// TIA Portal V20 export
// export: Created 2025-12-01T14:57:04.1801428Z, ExportSetting None, DisplayName Totally Integrated Automation Portal, DisplayVersion V20 Update 3, DisplayName TIA Portal Openness, DisplayVersion V20 Update 3, DisplayName TIA Portal Version Control Interface, DisplayVersion V20 Update 3, DisplayName STEP 7 Professional, DisplayVersion V20 Update 3, DisplayName STEP 7 Safety, DisplayVersion V20 Update 2, DisplayName WinCC Basic/Comfort/Advanced, DisplayVersion V20 Update 3, DisplayName WinCC Professional, DisplayVersion V20 Update 3, DisplayName WinCC Unified, DisplayVersion V20 Update 3
FUNCTION "FC762_EventosAlturaPedido" : Void   // FC762, STL
TITLE = Emision de los Eventos del la Etiquetadora
{ S7_Optimized_Access := 'FALSE' }
AUTHOR : TRACKING
NAME : 20141014
VERSION : 4.0
// stored: AutoNumber false
   VAR_INPUT
      NumMaquina : UInt;   // Numero de Maquina
      EstadoMaquina : "EstadoZona";   // Estado de la Maquina
      EstadoVIMaquina : "EstadoMaquina";   // Estado del VI de la Maquina
      AlturaPedido : UInt;   // Altura de la Paleta
      MaquinaDeJdT02 : Bool;
   END_VAR
   VAR_IN_OUT
      EnviarAlturaPedido : Bool;   // Enviar Evento
   END_VAR
   VAR_TEMP
      NumeroUT : UInt;
      McKey : UDInt;
      P_EmiEventos : DWord;
      DBEventos : Word;
      NumDBEventos : UInt;
      MaxBytes : UInt;
      NumBytes : UInt;
      OffsetInicial : UInt;
      OffsetFinal : UInt;
      Conversion : DWord;
      WordConvertir : Word;
      Valor : UDInt;
   END_VAR
BEGIN

NETWORK
TITLE = Inicializaciones
///////////////////////////////////////////////////////////////////////////////
/// Inicio --> Pertenece al JDT 02

      L     "JDT1_NDB_EventosEmi";
      T     #DBEventos;
      T     #NumDBEventos;
      L     "JDT1_MaxBytes";
      T     #MaxBytes;

      AN    #MaquinaDeJdT02;
      JC    NoJdT02;

      L     "JDT2_NDB_EventosEmi";
      T     #DBEventos;
      T     #NumDBEventos;
      L     "JDT2_MaxBytes";
      T     #MaxBytes;

NoJdT02:NOP   0;

/// Final --> Pertenece al JDT 02
///////////////////////////////////////////////////////////////////////////////



NETWORK
TITLE = Mirar si se pueden generar eventos
// - Inicializo el Numero de Bytes y el puntero del DB de Eventos Generados
// - Calcula el Tamaño de bytes que hay en el DB de Eventos Genardos
// - Comprobamos si hay sitio para Eventos
///////////////////////////////////////////////////////////////////////////////
// Inicializo el Numero de Bytes y el puntero del DB Eventos Generados

      L     0;
      T     #NumBytes;  // Inicializo el numero de Bytes
      LAR2;  // Inicializo el puntero de Eventos Generados

///////////////////////////////////////////////////////////////////////////////
// Calcula el tamaño de bytes que hay en el DB Eventos Generados

      OPN   DB [#DBEventos];

Inicio_BusquedaFinalEventos:NOP   0;
      L     DBB [AR2, P#0.0];
      L     0;
      ==I;
      JC    Ein_BusquedaFinalEventos;  // Buscamos el final del DB = 0

      +AR2  P#1.0;
      JU    Inicio_BusquedaFinalEventos;

Ein_BusquedaFinalEventos:NOP   0;
      TAR2;  // Guardo el puntero
      T     #P_EmiEventos;  // Sacamos el NumBytes Escritos
      SRD   3;
      T     #NumBytes;

///////////////////////////////////////////////////////////////////////////////
// Comprobamos si hay sitio para mas Eventos

      L     #NumBytes;  // Miramos si hay sitio
      L     #MaxBytes;  // Max. que se pueden emitir, parametro
      >I;
      JC    Final;  // No se pueden generar más eventos



NETWORK
TITLE = Distribucion
///////////////////////////////////////////////////////////////////////////////
// --- Distribucion  del Envio de la Altura de Paleta

      A     #EnviarAlturaPedido;  // Enviar la Altura ?
      JC    EmitirEvento;


///////////////////////////////////////////////////////////////////////////////
// --- Fin del Control

      JU    Final;



NETWORK
TITLE = Emision del Evento
EmitirEvento:NOP   0;

/////////////////////////////////////////////////////////////////////////////
// - Recoger Datos de la UT a Enviar (Primera de la Mesa)

      L     "DB810_ColasMesas".Colas[#NumMaquina].UT_PrimeraMesa;
      T     #NumeroUT;

      L     "DB812_UTs_Control".UT[#NumeroUT].Mckey;
      T     #McKey;

      L     #AlturaPedido;  //   Se guarda la Altura Enviada
      T     "DB815_UTs_Datos".UT[#NumeroUT].CotaAltura;


/////////////////////////////////////////////////////////////////////////////
// --- Formateo del Evento PROC - Estado del Proceso de la Maquina

      L     #P_EmiEventos;
      LAR2;  // Puntero al DB de Eventos Generados

      TAR2;  // Mirar si es el primer evento de la lista
      L     0;
      ==I;
      JC    NoEsInicio_ListaDeEventos;  // Es el primero

      OPN   DB [#DBEventos];
      L     ',';  // Separador entre eventos ','
      T     DBB [AR2, P#0.0];
      +AR2  P#1.0;

NoEsInicio_ListaDeEventos:NOP   0;
      OPN   DB [#DBEventos];  // DB de Eventos Generados (A Emitir)
      L     '{';  // Inicio de Evento '{'
      T     DBB [AR2, P#0.0];
      +AR2  P#1.0;


/////////////////////////////////////////////////////////////////////////////
// --- Cuerpo del Evento PROC

      L     'DATO';  // Evento 'DATO'
      T     DBD [AR2, P#0.0];
      +AR2  P#4.0;


// --- Escritura del Atributo MCKEY

      L     '[';  // Evento - Atributo MCKY '[MCKY]'
      T     DBB [AR2, P#0.0];
      L     'MCKY';
      T     DBD [AR2, P#1.0];
      L     ']';
      T     DBB [AR2, P#5.0];
      +AR2  P#6.0;

      TAR2;
      SRD   3;
      T     #OffsetInicial;  // Miro que offset tiene la String

      L     #McKey;
      T     #Valor;

      CALL  "FC893_Obtener_StringDelAtributo"
      ( DB_String := #NumDBEventos,
        OffsetIni := #OffsetInicial,
        Valor     := #Valor,
        OffsetFin := #OffsetFinal
      );  // Llamo a ObtenerStrinAtributo

      L     #OffsetFinal;
      SLD   3;
      LAR2;  // Recupero que offset tiene la String


/// --- Escritura del Atributo MESA

      OPN   DB [#DBEventos];  // DB de Eventos Generados (A Emitir)
      L     '[';  // Evento - Atributo MESA '[MESA]'
      T     DBB [AR2, P#0.0];
      L     'MESA';
      T     DBD [AR2, P#1.0];
      L     ']';
      T     DBB [AR2, P#5.0];
      +AR2  P#6.0;

      TAR2;
      SRD   3;
      T     #OffsetInicial;  // Miro que offset tiene la String

      L     "CTE_OffsetMesa";
      L     #NumMaquina;  // Numero de Maquina
      +I;
      T     #Valor;

      CALL  "FC893_Obtener_StringDelAtributo"
      ( DB_String := #NumDBEventos,
        OffsetIni := #OffsetInicial,
        Valor     := #Valor,
        OffsetFin := #OffsetFinal
      );  // Llamo a ObtenerStrinAtributo

      L     #OffsetFinal;
      SLD   3;
      LAR2;  // Recupero que offset tiene la String


// --- Escritura del Atributo 'COTA'

      OPN   DB [#DBEventos];
      L     '[';  // Evento - Atributo Altura Cota '[COTA]'
      T     DBB [AR2, P#0.0];
      L     'COTA';
      T     DBD [AR2, P#1.0];
      L     ']';
      T     DBB [AR2, P#5.0];
      +AR2  P#6.0;


      TAR2;  // Escritura del Atributo
      SRD   3;
      T     #OffsetInicial;  // Miro que offset tiene la String

      L     #AlturaPedido;
      T     #Valor;

      CALL  "FC893_Obtener_StringDelAtributo"
      ( DB_String := #NumDBEventos,
        OffsetIni := #OffsetInicial,
        Valor     := #Valor,
        OffsetFin := #OffsetFinal
      );  // Llamo a ObtenerStrinAtributo

      L     #OffsetFinal;
      SLD   3;
      LAR2;  // Recupero que offset tiene la String


/////////////////////////////////////////////////////////////////////////////
// --- Final del formateo del Evento

      OPN   DB [#DBEventos];  // DB de Eventos Generados (A Emitir)
      L     '}';  // Fin de Evento '}'
      T     DBB [AR2, P#0.0];
      +AR2  P#1.0;


/////////////////////////////////////////////////////////////////////////////
// --- Dar por formateado el Evento
      SET;
      R     #EnviarAlturaPedido;

      JU    Final;  // Ya se ha generado el evento de la Maquina

// --- Fin del Formateo del Evento de Estado del Proceso
/////////////////////////////////////////////////////////////////////////////



NETWORK
TITLE = Fin de la Funcion
///////////////////////////////////////////////////////////////////////////////
// --- Final de la función
Final:NOP   0;



END_FUNCTION
